(* CODESYS project assemblyAndPackoutCell.export

Project tree, tasks and I/O mapping:
  Device : CODESYS Control Win V3 x64, CODESYS, version 3.5.22.30
    application Application
      libraries: Standard, 3.5.22.0 (System)
      task MainTask (cyclic, interval t#20ms, priority 1) calls PLC_PRG
      data type E_AssemblerState
      global variables AssemblyConstants
      global variables Commands
      global variables FIO
      function block FB_AssemblerCell [ST]
      function block FB_OperatorControl [ST]
      program PLC_PRG [ST]
      Symbols
*)

// Device/Application/E_AssemblerState
TYPE E_AssemblerState :
(
    Stopped                := 0,
    Homing                 := 10,
    WaitingForParts        := 20,
    ClampingParts          := 30,
    LoweringToLid          := 40,
    GrippingLid            := 50,
    ReleasingLidClamp      := 60,
    RaisingLid             := 70,
    MovingToBase           := 80,
    LoweringToBase         := 90,
    ReleasingLid           := 100,
    RaisingFromBase        := 110,
    ReturningHome          := 120,
    ReleasingProduct       := 130,
    WaitingForProductExit  := 140,
    Faulted                := 900
);
END_TYPE

// Device/Application/AssemblyConstants
VAR_GLOBAL CONSTANT

    tAssemblerClampTimeout       : TIME := T#5S;
    tAssemblerFeedTimeout        : TIME := T#15S;
    tAssemblerGrabSettle         : TIME := T#300MS;
    tAssemblerHomeSettle         : TIME := T#500MS;
    tAssemblerMotionTimeout      : TIME := T#5S;
    tAssemblerProductExitTimeout : TIME := T#10S;
    tAssemblerReleaseSettle      : TIME := T#300MS;

END_VAR

// Device/Application/Commands
VAR_GLOBAL

    // Momentary commissioning commands.
    // Pulse TRUE and then return to FALSE.

    xResetPB : BOOL;
    xStartPB : BOOL;
    xStopPB  : BOOL;

END_VAR

// Device/Application/FIO
VAR_GLOBAL

    // =========================================================
    // FACTORY I/O SENSORS
    // Factory I/O -> PLC
    // =========================================================

    rFactoryIOTimeScale       : REAL; // FACTORY I/O (Time Scale)

    xAutoModeSelected         : BOOL; // Auto
    xBaseAtPlace              : BOOL; // Base at place
    xBaseClamped              : BOOL; // Base clamped
    xBasesPositionerAtLimit   : BOOL; // Pos. at limit (bases)
    xEmergencyStop            : BOOL; // Emergency stop
    xFactoryIOPaused          : BOOL; // FACTORY I/O (Paused)
    xFactoryIOReset           : BOOL; // FACTORY I/O (Reset)
    xFactoryIORunning         : BOOL; // FACTORY I/O (Running)
    xItemDetected             : BOOL; // Item detected
    xLidAtPlace               : BOOL; // Lid at place
    xLidClamped               : BOOL; // Lid clamped
    xManualModeSelected       : BOOL; // Manual
    xMovingX                  : BOOL; // Moving X
    xMovingZ                  : BOOL; // Moving Z
    xPartLeaving              : BOOL; // Part leaving
    xResetPB                  : BOOL; // Reset
    xStartPB                  : BOOL; // Start
    xStopPB                   : BOOL; // Stop


    // =========================================================
    // FACTORY I/O ACTUATORS
    // PLC -> Factory I/O
    // =========================================================

    diFactoryIOCameraPositionCmd : DINT; // FACTORY I/O (Camera Position)
    diProductCounterDisplay      : DINT; // Counter

    xBaseClampCmd                : BOOL; // Clamp base
    xBasesConveyorCmd            : BOOL; // Bases conveyor
    xBasesEmitterCmd             : BOOL; // Bases emitter
    xBasesPositionerRaiseCmd     : BOOL; // Pos. raise (bases)
    xFactoryIOPauseCmd           : BOOL; // FACTORY I/O (Pause)
    xFactoryIOResetCmd           : BOOL; // FACTORY I/O (Reset)
    xFactoryIORunCmd             : BOOL; // FACTORY I/O (Run)
    xFinishedProductRemoverCmd   : BOOL; // Remover 1
    xGrabCmd                     : BOOL; // Grab
    xLidClampCmd                 : BOOL; // Clamp lid
    xLidsConveyorCmd             : BOOL; // Lids conveyor
    xLidsEmitterCmd              : BOOL; // Lids emitter
    xLidsPositionerRaiseCmd      : BOOL; // Pos. raise (lids)
    xMoveXCmd                    : BOOL; // Move X
    xMoveZCmd                    : BOOL; // Move Z
    xResetLightCmd               : BOOL; // Reset light
    xStartLightCmd               : BOOL; // Start light
    xStopLightCmd                : BOOL; // Stop light
    xUnusedLidRemoverCmd         : BOOL; // Remover 2

END_VAR

// Device/Application/PLC_PRG
PROGRAM PLC_PRG
VAR
    diProductsCompleted : DINT;

    eAssemblerState : E_AssemblerState;

    fbAssemblerCell : FB_AssemblerCell;
    fbOperator      : FB_OperatorControl;

    uiAssemblerFaultCode : UINT;

    xAssemblerBusy             : BOOL;
    xAssemblerFaulted          : BOOL;
    xAssemblerReady            : BOOL;
    xBaseClampCmd              : BOOL;
    xBasesConveyorCmd          : BOOL;
    xBasesPositionerRaiseCmd   : BOOL;
    xEnableAutomatic           : BOOL;
    xGrabCmd                   : BOOL;
    xLidClampCmd               : BOOL;
    xLidsConveyorCmd           : BOOL;
    xMoveXCmd                  : BOOL;
    xMoveZCmd                  : BOOL;
    xPlantFaulted              : BOOL;
    xProductCompletePulse      : BOOL;
	xRecoveryResetRequired 	   : BOOL;
    xResetPulse                : BOOL;
    xResetRequired             : BOOL;
    xRunLatched                : BOOL;
	xStopPending 			   : BOOL;
END_VAR

// =============================================================
// 1. PLANT FAULT STATUS FROM THE PREVIOUS PLC SCAN
// =============================================================

xPlantFaulted :=
    xAssemblerFaulted;

// =============================================================
// 2. OPERATOR CONTROL
// Commands may originate from either CODESYS commissioning
// variables or the physical Factory I/O control panel.
// =============================================================

// Preserve the pre-reset recovery requirement for this scan.
xRecoveryResetRequired :=
xResetRequired;

fbOperator(
    xAutoModeSelected :=
        FIO.xAutoModeSelected,

    xEmergencyStop :=
        NOT FIO.xEmergencyStop,

    xFactoryIOPaused :=
        FIO.xFactoryIOPaused,

    xFactoryIORunning :=
        FIO.xFactoryIORunning,

    xManualModeSelected :=
        FIO.xManualModeSelected,

    xPlantFaulted :=
        xPlantFaulted,

    xResetPB :=
        Commands.xResetPB
        OR FIO.xFactoryIOReset
        OR FIO.xResetPB,

	xSafeToStop :=
		xProductCompletePulse,
		
    xStartPB :=
        Commands.xStartPB
        OR FIO.xStartPB,

    xStopPB :=
        Commands.xStopPB
        OR NOT FIO.xStopPB,

    xEnableAutomatic =>
        xEnableAutomatic,

    xResetPulse =>
        xResetPulse,

    xResetRequired =>
        xResetRequired,

    xRunLatched =>
        xRunLatched,
		
	xStopPending =>
    	xStopPending
);

// =============================================================
// 3. ASSEMBLER CELL
// =============================================================

fbAssemblerCell(
    tClampTimeout :=
        AssemblyConstants.tAssemblerClampTimeout,

    tFeedTimeout :=
        AssemblyConstants.tAssemblerFeedTimeout,

    tGrabSettle :=
        AssemblyConstants.tAssemblerGrabSettle,

    tHomeSettle :=
        AssemblyConstants.tAssemblerHomeSettle,

    tMotionTimeout :=
        AssemblyConstants.tAssemblerMotionTimeout,

    tProductExitTimeout :=
        AssemblyConstants.tAssemblerProductExitTimeout,

    tReleaseSettle :=
        AssemblyConstants.tAssemblerReleaseSettle,

    xBaseAtPlace :=
        FIO.xBaseAtPlace,

    xBaseClamped :=
        FIO.xBaseClamped,

    xBasesPositionerAtLimit :=
        FIO.xBasesPositionerAtLimit,

    xEnable :=
        xEnableAutomatic,

    xItemDetected :=
        FIO.xItemDetected,

    xLidAtPlace :=
        FIO.xLidAtPlace,

    xLidClamped :=
        FIO.xLidClamped,

    xMovingX :=
        FIO.xMovingX,

    xMovingZ :=
        FIO.xMovingZ,

    xPartLeaving :=
        FIO.xPartLeaving,

    xReset :=
        xResetPulse,

    diProductsCompleted =>
        diProductsCompleted,

    eState =>
        eAssemblerState,

    uiFaultCode =>
        uiAssemblerFaultCode,

    xBaseClampCmd =>
        xBaseClampCmd,

    xBasesConveyorCmd =>
        xBasesConveyorCmd,

    xBasesPositionerRaiseCmd =>
        xBasesPositionerRaiseCmd,

    xBusy =>
        xAssemblerBusy,

    xFaulted =>
        xAssemblerFaulted,

    xGrabCmd =>
        xGrabCmd,

    xLidClampCmd =>
        xLidClampCmd,

    xLidsConveyorCmd =>
        xLidsConveyorCmd,

    xMoveXCmd =>
        xMoveXCmd,

    xMoveZCmd =>
        xMoveZCmd,

    xProductCompletePulse =>
        xProductCompletePulse,

    xReady =>
        xAssemblerReady
);

// =============================================================
// 4. FACTORY I/O OUTPUT BOUNDARY
// =============================================================
// -------------------------------------------------------------
// Assembly equipment
// -------------------------------------------------------------

FIO.xBaseClampCmd :=
    xBaseClampCmd;

FIO.xBasesConveyorCmd :=
    xBasesConveyorCmd;

FIO.xBasesPositionerRaiseCmd :=
    xBasesPositionerRaiseCmd;

FIO.xGrabCmd :=
    xGrabCmd;

FIO.xLidClampCmd :=
    xLidClampCmd;

FIO.xLidsConveyorCmd :=
    xLidsConveyorCmd;

FIO.xLidsPositionerRaiseCmd :=
	FALSE;

FIO.xMoveXCmd :=
    xMoveXCmd;

FIO.xMoveZCmd :=
    xMoveZCmd;

// -------------------------------------------------------------
// Emitters and removers
// -------------------------------------------------------------

FIO.xBasesEmitterCmd :=
    xEnableAutomatic;

FIO.xFinishedProductRemoverCmd :=
    xEnableAutomatic;

FIO.xLidsEmitterCmd :=
    xEnableAutomatic;

FIO.xUnusedLidRemoverCmd :=
    xEnableAutomatic;

// -------------------------------------------------------------
// Control-panel lights
// -------------------------------------------------------------

FIO.xResetLightCmd :=
    xResetRequired
    OR xAssemblerFaulted;

FIO.xStartLightCmd :=
    xEnableAutomatic
	AND NOT xStopPending;

FIO.xStopLightCmd :=
    NOT xRunLatched
	OR xStopPending;

// -------------------------------------------------------------
// Product counter display
// -------------------------------------------------------------

FIO.diProductCounterDisplay :=
    diProductsCompleted;

// -------------------------------------------------------------
// Factory I/O simulation controls
// Run, Pause and Camera remain manually controlled.
// The physical scene resets only during abnormal recovery.
// -------------------------------------------------------------

FIO.diFactoryIOCameraPositionCmd :=
    0;

FIO.xFactoryIOPauseCmd :=
    FALSE;

FIO.xFactoryIOResetCmd :=
    xResetPulse
    AND xRecoveryResetRequired;

FIO.xFactoryIORunCmd :=
    FALSE;

END_PROGRAM

// Device/Application/FB_AssemblerCell
FUNCTION_BLOCK FB_AssemblerCell
VAR_INPUT
    tClampTimeout       : TIME;
    tFeedTimeout        : TIME;
    tGrabSettle         : TIME;
    tHomeSettle         : TIME;
    tMotionTimeout      : TIME;
    tProductExitTimeout : TIME;
    tReleaseSettle      : TIME;

    xBaseAtPlace            : BOOL;
    xBaseClamped            : BOOL;
    xBasesPositionerAtLimit : BOOL;
    xEnable                 : BOOL;
    xItemDetected           : BOOL;
    xLidAtPlace             : BOOL;
    xLidClamped             : BOOL;
    xMovingX                : BOOL;
    xMovingZ                : BOOL;
    xPartLeaving            : BOOL;
    xReset                  : BOOL;
END_VAR

VAR_OUTPUT
    diProductsCompleted : DINT;
    eState              : E_AssemblerState;
    uiFaultCode         : UINT;

    xBaseClampCmd            : BOOL;
    xBasesConveyorCmd        : BOOL;
    xBasesPositionerRaiseCmd : BOOL;
    xBusy                    : BOOL;
    xFaulted                 : BOOL;
    xGrabCmd                 : BOOL;
    xLidClampCmd             : BOOL;
    xLidsConveyorCmd         : BOOL;
    xMoveXCmd                : BOOL;
    xMoveZCmd                : BOOL;
    xProductCompletePulse    : BOOL;
    xReady                   : BOOL;
END_VAR

VAR
    ePreviousState : E_AssemblerState :=
        E_AssemblerState.Stopped;

    fbClampTimeout       : TON;
    fbFeedTimeout        : TON;
    fbGrabSettle         : TON;
    fbGrabTimeout        : TON;
    fbHomeSettle         : TON;
    fbMotionTimeout      : TON;
    fbProductExitTimeout : TON;
    fbReleaseSettle      : TON;

    rtPartLeaving : R_TRIG;

    xMotionObserved : BOOL;
    xStateChanged   : BOOL;
END_VAR

// =============================================================
// DEFAULT COMMANDS
//
// Every command must be deliberately enabled by the active state.
// =============================================================

xBaseClampCmd := FALSE;
xBasesConveyorCmd := FALSE;
xBasesPositionerRaiseCmd := FALSE;
xGrabCmd := FALSE;
xLidClampCmd := FALSE;
xLidsConveyorCmd := FALSE;
xMoveXCmd := FALSE;
xMoveZCmd := FALSE;
xProductCompletePulse := FALSE;

// =============================================================
// EDGE AND STATE-ENTRY DETECTION
// =============================================================

rtPartLeaving(CLK := xPartLeaving);

xStateChanged :=
    eState <> ePreviousState;

IF xStateChanged THEN
    ePreviousState := eState;
    xMotionObserved := FALSE;
END_IF;

// =============================================================
// STATE TIMERS
// =============================================================

fbClampTimeout(
    IN :=
        xEnable
        AND NOT xStateChanged
        AND (
            (eState = E_AssemblerState.ClampingParts)
            OR
            (eState = E_AssemblerState.ReleasingLidClamp)
        ),
    PT := tClampTimeout
);

fbFeedTimeout(
    IN :=
        xEnable
        AND NOT xStateChanged
        AND (eState = E_AssemblerState.WaitingForParts),
    PT := tFeedTimeout
);

fbGrabSettle(
    IN :=
        xEnable
        AND (eState = E_AssemblerState.GrippingLid)
        AND xItemDetected,
    PT := tGrabSettle
);

fbGrabTimeout(
    IN :=
        xEnable
        AND NOT xStateChanged
        AND (eState = E_AssemblerState.GrippingLid),
    PT := tMotionTimeout
);

fbHomeSettle(
    IN :=
        xEnable
        AND (eState = E_AssemblerState.Homing)
        AND NOT xMovingX
        AND NOT xMovingZ,
    PT := tHomeSettle
);

fbMotionTimeout(
    IN :=
        xEnable
        AND NOT xStateChanged
        AND (
            (eState = E_AssemblerState.Homing)
            OR
            (eState = E_AssemblerState.LoweringToLid)
            OR
            (eState = E_AssemblerState.LoweringToBase)
            OR
            (eState = E_AssemblerState.MovingToBase)
            OR
            (eState = E_AssemblerState.RaisingFromBase)
            OR
            (eState = E_AssemblerState.RaisingLid)
            OR
            (eState = E_AssemblerState.ReturningHome)
			OR
			(eState = E_AssemblerState.ReleasingProduct)
        ),
    PT := tMotionTimeout
);	

fbProductExitTimeout(
    IN :=
        xEnable
        AND NOT xStateChanged
        AND (eState = E_AssemblerState.WaitingForProductExit),
    PT := tProductExitTimeout
);

fbReleaseSettle(
    IN :=
        xEnable
        AND (eState = E_AssemblerState.ReleasingLid),
    PT := tReleaseSettle
);

// =============================================================
// RESET AND DISABLED CONDITIONS
// =============================================================

IF xReset THEN

    diProductsCompleted := 0;
    eState := E_AssemblerState.Stopped;
    uiFaultCode := 0;
    xMotionObserved := FALSE;

ELSIF NOT xEnable THEN

    // Fault state remains latched until Reset.
    IF eState <> E_AssemblerState.Faulted THEN
        eState := E_AssemblerState.Stopped;
    END_IF;

// =============================================================
// AUTOMATIC ASSEMBLY SEQUENCE
// =============================================================

ELSE

    CASE eState OF

        // -----------------------------------------------------
        // Begin every enabled run by returning the arm to its
        // default raised position above the lid.
        // -----------------------------------------------------

        E_AssemblerState.Stopped:

            eState := E_AssemblerState.Homing;

        // -----------------------------------------------------
        // Move X = FALSE: above the lid.
        // Move Z = FALSE: raised.
        //
        // The settle timer also handles the case where the arm
        // was already home and therefore produces no movement.
        // -----------------------------------------------------

        E_AssemblerState.Homing:

            IF fbHomeSettle.Q THEN
                eState := E_AssemblerState.WaitingForParts;

            ELSIF fbMotionTimeout.Q THEN
                uiFaultCode := 201;
                eState := E_AssemblerState.Faulted;
            END_IF;

        // -----------------------------------------------------
        // Keeps both positioners lowered while feeding material.
        // Each conveyor stops independently when its part
        // reaches the assembly position.
        // -----------------------------------------------------

		E_AssemblerState.WaitingForParts:
		
			// Keep both positioning assemblies lowered.
			// Feed each conveyor independently until its part arrives.
		
			xBasesConveyorCmd := NOT xBaseAtPlace;
			xLidsConveyorCmd := NOT xLidAtPlace;
		
			IF xBaseAtPlace
			AND xLidAtPlace THEN
		
				eState := E_AssemblerState.ClampingParts;
		
			ELSIF fbFeedTimeout.Q THEN
				uiFaultCode := 101;
				eState := E_AssemblerState.Faulted;
			END_IF;

        // -----------------------------------------------------
        // Secure both parts before the picker moves.
        // -----------------------------------------------------

        E_AssemblerState.ClampingParts:

			// Continue conveying each detected part into its clamp.
			// Stop each conveyor independently once clamped.
		
			xBaseClampCmd := TRUE;
			xBasesConveyorCmd := NOT xBaseClamped;
			xLidClampCmd := TRUE;
			xLidsConveyorCmd := NOT xLidClamped;
		
			IF xBaseClamped
			AND xLidClamped THEN
		
				eState := E_AssemblerState.LoweringToLid;
		
			ELSIF fbClampTimeout.Q THEN
				uiFaultCode := 102;
				eState := E_AssemblerState.Faulted;
			END_IF;

        // -----------------------------------------------------
        // Lower the picker onto the clamped lid.
        // -----------------------------------------------------

        E_AssemblerState.LoweringToLid:

            xBaseClampCmd := TRUE;
            
            xLidClampCmd := TRUE;
            
            xMoveZCmd := TRUE;

            IF xMovingZ THEN
                xMotionObserved := TRUE;
            END_IF;

            IF xMotionObserved AND NOT xMovingZ THEN
                eState := E_AssemblerState.GrippingLid;

            ELSIF fbMotionTimeout.Q THEN
                uiFaultCode := 202;
                eState := E_AssemblerState.Faulted;
            END_IF;

        // -----------------------------------------------------
        // Energise the suction cup and confirm the lid.
        // -----------------------------------------------------

        E_AssemblerState.GrippingLid:

            xBaseClampCmd := TRUE;
            
            xGrabCmd := TRUE;
            xLidClampCmd := TRUE;
            
            xMoveZCmd := TRUE;

            IF fbGrabSettle.Q THEN
                eState := E_AssemblerState.ReleasingLidClamp;

            ELSIF fbGrabTimeout.Q THEN
                uiFaultCode := 203;
                eState := E_AssemblerState.Faulted;
            END_IF;

        // -----------------------------------------------------
        // Release the lid clamp while suction retains the lid.
        // -----------------------------------------------------

        E_AssemblerState.ReleasingLidClamp:

            xBaseClampCmd := TRUE;
            
            xGrabCmd := TRUE;
            
            xMoveZCmd := TRUE;

            IF NOT xLidClamped THEN
                eState := E_AssemblerState.RaisingLid;

            ELSIF fbClampTimeout.Q THEN
                uiFaultCode := 204;
                eState := E_AssemblerState.Faulted;
            END_IF;

        // -----------------------------------------------------
        // Raise the collected lid.
        // -----------------------------------------------------

        E_AssemblerState.RaisingLid:

            xBaseClampCmd := TRUE;
            
            xGrabCmd := TRUE;
            

            IF xMovingZ THEN
                xMotionObserved := TRUE;
            END_IF;

            IF xMotionObserved AND NOT xMovingZ THEN
                eState := E_AssemblerState.MovingToBase;

            ELSIF fbMotionTimeout.Q THEN
                uiFaultCode := 205;
                eState := E_AssemblerState.Faulted;
            END_IF;

        // -----------------------------------------------------
        // Transfer from the home position above the lid to the
        // assembly position above the base.
        // -----------------------------------------------------

        E_AssemblerState.MovingToBase:

            xBaseClampCmd := TRUE;
            
            xGrabCmd := TRUE;
            
            xMoveXCmd := TRUE;

            IF xMovingX THEN
                xMotionObserved := TRUE;
            END_IF;

            IF xMotionObserved AND NOT xMovingX THEN
                eState := E_AssemblerState.LoweringToBase;

            ELSIF fbMotionTimeout.Q THEN
                uiFaultCode := 206;
                eState := E_AssemblerState.Faulted;
            END_IF;

        // -----------------------------------------------------
        // Lower the lid onto the clamped base.
        // -----------------------------------------------------

        E_AssemblerState.LoweringToBase:

            xBaseClampCmd := TRUE;
            
            xGrabCmd := TRUE;
            
            xMoveXCmd := TRUE;
            xMoveZCmd := TRUE;

            IF xMovingZ THEN
                xMotionObserved := TRUE;
            END_IF;

            IF xMotionObserved AND NOT xMovingZ THEN
                eState := E_AssemblerState.ReleasingLid;

            ELSIF fbMotionTimeout.Q THEN
                uiFaultCode := 207;
                eState := E_AssemblerState.Faulted;
            END_IF;

        // -----------------------------------------------------
        // Release suction. Correct physical alignment causes
        // Factory I/O to join the lid and base automatically.
        // -----------------------------------------------------

        E_AssemblerState.ReleasingLid:

            xBaseClampCmd := TRUE;
            
            
            xMoveXCmd := TRUE;
            xMoveZCmd := TRUE;

            IF fbReleaseSettle.Q THEN
                eState := E_AssemblerState.RaisingFromBase;
            END_IF;

        // -----------------------------------------------------
        // Raise clear of the assembled product.
        // -----------------------------------------------------

        E_AssemblerState.RaisingFromBase:

            xBaseClampCmd := TRUE;
            
            
            xMoveXCmd := TRUE;

            IF xMovingZ THEN
                xMotionObserved := TRUE;
            END_IF;

            IF xMotionObserved AND NOT xMovingZ THEN
                eState := E_AssemblerState.ReturningHome;

            ELSIF fbMotionTimeout.Q THEN
                uiFaultCode := 208;
                eState := E_AssemblerState.Faulted;
            END_IF;

        // -----------------------------------------------------
        // Return to the default position above the lid.
        // -----------------------------------------------------

        E_AssemblerState.ReturningHome:

            xBaseClampCmd := TRUE;
            
            

            IF xMovingX THEN
                xMotionObserved := TRUE;
            END_IF;

            IF xMotionObserved AND NOT xMovingX THEN
                eState := E_AssemblerState.ReleasingProduct;

            ELSIF fbMotionTimeout.Q THEN
                uiFaultCode := 209;
                eState := E_AssemblerState.Faulted;
            END_IF;

        // -----------------------------------------------------
        // Release the base clamp and raise the base positioner.
        // The finished product exits along the base conveyor.
        // -----------------------------------------------------

        E_AssemblerState.ReleasingProduct:

			// Release the base clamp through its default FALSE command
			// and raise the positioning assembly clear of the product.
		
			xBasesPositionerRaiseCmd := TRUE;
		
			IF xBasesPositionerAtLimit THEN
				eState := E_AssemblerState.WaitingForProductExit;
		
			ELSIF fbMotionTimeout.Q THEN
				uiFaultCode := 210; // Base positioner failed to raise.
				eState := E_AssemblerState.Faulted;
			END_IF;

        // -----------------------------------------------------
        // Wait for the downstream sensor. Its rising edge gives
        // exactly one count for each completed product.
        // -----------------------------------------------------

        E_AssemblerState.WaitingForProductExit:

			// Once clearance has been confirmed, keep the conveyors
			// running without continuously depending on the limit signal.
		
			xBasesConveyorCmd := TRUE;
			xBasesPositionerRaiseCmd := TRUE;
			xLidsConveyorCmd := NOT xLidAtPlace;
		
			IF rtPartLeaving.Q THEN
		
				diProductsCompleted :=
					diProductsCompleted + 1;
		
				xProductCompletePulse := TRUE;
				eState := E_AssemblerState.WaitingForParts;
		
			ELSIF fbMotionTimeout.Q THEN
				uiFaultCode := 301;
				eState := E_AssemblerState.Faulted;
			END_IF;

        // -----------------------------------------------------
        // Latched safe state.
        // -----------------------------------------------------

        E_AssemblerState.Faulted:

        // -----------------------------------------------------
        // Corrupted or unexpected enumeration value.
        // -----------------------------------------------------

        ELSE

            uiFaultCode := 999;
            eState := E_AssemblerState.Faulted;

    END_CASE;

END_IF;

// =============================================================
// STATUS OUTPUTS
// =============================================================

xFaulted :=
    eState = E_AssemblerState.Faulted;

xReady :=
    xEnable
    AND (eState = E_AssemblerState.WaitingForParts);

xBusy :=
    xEnable
    AND (eState <> E_AssemblerState.Stopped)
    AND (eState <> E_AssemblerState.WaitingForParts)
    AND (eState <> E_AssemblerState.Faulted);

// Ensure every physical command is de-energised after a fault.
IF xFaulted THEN
    xBaseClampCmd := FALSE;
    xBasesConveyorCmd := FALSE;
    xBasesPositionerRaiseCmd := FALSE;
    xGrabCmd := FALSE;
    xLidClampCmd := FALSE;
    xLidsConveyorCmd := FALSE;
    xMoveXCmd := FALSE;
    xMoveZCmd := FALSE;
END_IF;

END_FUNCTION_BLOCK

// Device/Application/FB_OperatorControl
FUNCTION_BLOCK FB_OperatorControl
VAR_INPUT
    xAutoModeSelected   : BOOL;
    xEmergencyStop      : BOOL;
    xFactoryIOPaused    : BOOL;
    xFactoryIORunning   : BOOL;
    xManualModeSelected : BOOL;
    xPlantFaulted       : BOOL;
    xResetPB            : BOOL;
	xSafeToStop 		: BOOL;
    xStartPB            : BOOL;
    xStopPB             : BOOL;
END_VAR

VAR_OUTPUT
    xEnableAutomatic : BOOL;
    xResetPulse      : BOOL;
    xResetRequired   : BOOL;
    xRunLatched      : BOOL;
	xStopPending 	 : BOOL;
END_VAR

VAR
    rtReset        : R_TRIG;
    rtStart        : R_TRIG;
    rtStop         : R_TRIG;
    xAutoModeValid : BOOL;
END_VAR

// =============================================================
// EDGE DETECTION
// =============================================================

rtReset(CLK := xResetPB);
rtStart(CLK := xStartPB);
rtStop(CLK := xStopPB);

// =============================================================
// OPERATING-MODE VALIDATION
//
// Exactly one selector position must be active.
// =============================================================

xAutoModeValid :=
    xAutoModeSelected
    AND NOT xManualModeSelected;

// Reset is a one-scan event.
xResetPulse := FALSE;

// =============================================================
// OPERATOR COMMAND PRIORITIES
// =============================================================

IF xEmergencyStop THEN

    // Reset cannot bypass an active emergency stop.
    xResetRequired := TRUE;
    xRunLatched := FALSE;
    xStopPending := FALSE;

ELSIF rtReset.Q THEN

    // Reset clears latched faults but does not restart the plant.
    xResetPulse := TRUE;
    xResetRequired := FALSE;
    xRunLatched := FALSE;
    xStopPending := FALSE;

ELSIF xPlantFaulted THEN

    xResetRequired := TRUE;
    xRunLatched := FALSE;
    xStopPending := FALSE;

ELSIF NOT xAutoModeValid THEN

    xRunLatched := FALSE;
    xStopPending := FALSE;

ELSIF rtStop.Q THEN

    // Request a controlled stop. Automatic operation remains
	// enabled until the current product reaches the safe boundary.
	// A subsequent Start may resume without Reset.
    IF xSafeToStop THEN
        xRunLatched := FALSE;
        xStopPending := FALSE;
    ELSE
        xStopPending := TRUE;
    END_IF;

ELSIF xStopPending AND xSafeToStop THEN

    xRunLatched := FALSE;
    xStopPending := FALSE;

ELSIF rtStart.Q
AND xFactoryIORunning
AND NOT xFactoryIOPaused
AND NOT xResetRequired THEN

    xRunLatched := TRUE;
    xStopPending := FALSE;

END_IF;

// =============================================================
// FINAL AUTOMATIC-SEQUENCE PERMISSION
// =============================================================

xEnableAutomatic :=
    xRunLatched
    AND xAutoModeValid
    AND xFactoryIORunning
    AND NOT xEmergencyStop
    AND NOT xFactoryIOPaused
    AND NOT xPlantFaulted
    AND NOT xResetRequired;

END_FUNCTION_BLOCK
